FUNCTION_BLOCK UT_NumericValueInputMapping (* Service Interface Function Block Type *)
  (* Standard: ISO 11783-6; Classification: Input Number – ISO 11783-6; Function: All Inputs; Type: UT according to ISO 11783-6; Description: this maps to IUDINT *)
  (* Version 1.0, 2018-12-05, Jose Cabral *)
  (* Version 1.1, 2022-08-04, Franz Höpfinger, HR Agrartechnik GmbH *)
  (* Version 1.2, 2023-01-05, Franz Höpfinger, HR Agrartechnik GmbH *)
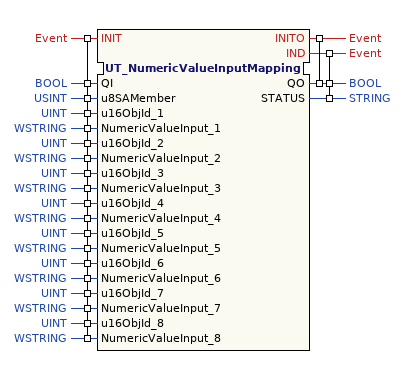
  EVENT_INPUT
    INIT WITH QI, u8SAMember, u16ObjId_1, NumericValueInput_1, u16ObjId_2, NumericValueInput_2, u16ObjId_3, NumericValueInput_3, u16ObjId_4, NumericValueInput_4, u16ObjId_5, NumericValueInput_5, u16ObjId_6, NumericValueInput_6, u16ObjId_7, NumericValueInput_7, u16ObjId_8, NumericValueInput_8; (* Service Initialization *)
  END_EVENT
  EVENT_OUTPUT
    INITO WITH QO; (* Initialization Confirm *)
    IND WITH QO, STATUS; (* Indication from Resource *)
  END_EVENT
  VAR_INPUT
    QI : BOOL; (* Event Input Qualifier *)
    u8SAMember : USINT := 255; (* Dummy !, set to 255 if in doubt. 0 deactivates FB. *)
    u16ObjId_1 : UINT := 21000; (* Object ID of Input 1 *)
    NumericValueInput_1 : WSTRING := "NumericValueInput_21000"; (* Identifier for Input 1 *)
    u16ObjId_2 : UINT := 21001; (* Object ID of Input 2 *)
    NumericValueInput_2 : WSTRING := "NumericValueInput_21001"; (* Identifier for Input 2 *)
    u16ObjId_3 : UINT := 21002; (* Object ID of Input 3 *)
    NumericValueInput_3 : WSTRING := "NumericValueInput_21002"; (* Identifier for Input 3 *)
    u16ObjId_4 : UINT := 21003; (* Object ID of Input 4 *)
    NumericValueInput_4 : WSTRING := "NumericValueInput_21003"; (* Identifier for Input 4 *)
    u16ObjId_5 : UINT := 21004; (* Object ID of Input 5 *)
    NumericValueInput_5 : WSTRING := "NumericValueInput_21004"; (* Identifier for Input 5 *)
    u16ObjId_6 : UINT := 21005; (* Object ID of Input 6 *)
    NumericValueInput_6 : WSTRING := "NumericValueInput_21005"; (* Identifier for Input 6 *)
    u16ObjId_7 : UINT := 21006; (* Object ID of Input 7 *)
    NumericValueInput_7 : WSTRING := "NumericValueInput_21006"; (* Identifier for Input 7 *)
    u16ObjId_8 : UINT := 21007; (* Object ID of Input 8 *)
    NumericValueInput_8 : WSTRING := "NumericValueInput_21007"; (* Identifier for Input 8 *)
  END_VAR
  VAR_OUTPUT
    QO : BOOL; (* Event Output Qualifier *)
    STATUS : STRING; (* Service Status *)
  END_VAR
END_FUNCTION_BLOCK
